(* TLS/PSK configuration *)
{attribute 'no_explicit_call':='Direct call not allowed for type FB_TlsConfig'}
{attribute 'no_assign'}
FUNCTION_BLOCK FB_TlsConfig
VAR
	_pskKey       : ARRAY[0..TCPADS_TLS_MAX_PSK_KEY_SIZE] OF BYTE;
	_pskKeyLen    : UDINT:=0;
	_sIdentity    : STRING(TCPADS_TLS_PSK_IDENTITY_SIZE);
	_sCaPath      : STRING(TCPADS_TLS_CERTIFICATE_PATH_SIZE);
	_sCrlPath     : STRING(TCPADS_TLS_CERTIFICATE_PATH_SIZE);
	_sCertPath    : STRING(TCPADS_TLS_CERTIFICATE_PATH_SIZE);
	_sKeyPath     : STRING(TCPADS_TLS_CERTIFICATE_PATH_SIZE);
	_sKeyPwd      : STRING(TCPADS_TLS_KEY_PASSWORD_SIZE);
	_listenFlags  : ST_TlsListenFlags:=DEFAULT_TLSLISTENFLAGS;
	_connectFlags : ST_TlsConnectFlags:=DEFAULT_TLSCONNECTFLAGS;
END_VAR

(* Adds CA certificate path *)
METHOD FINAL AddCa
VAR_INPUT
	sCaPath : STRING(TCPADS_TLS_CERTIFICATE_PATH_SIZE);
END_VAR
_sCaPath:=sCaPath;
END_METHOD

(* Adds certificate path *)
METHOD FINAL AddCert
VAR_INPUT
	sCertPath: STRING(TCPADS_TLS_CERTIFICATE_PATH_SIZE);
	sKeyPath: STRING(TCPADS_TLS_CERTIFICATE_PATH_SIZE);
	sKeyPwd: STRING(TCPADS_TLS_KEY_PASSWORD_SIZE);
END_VAR
_sCertPath:=sCertPath;
_sKeyPath:=sKeyPath;
_sKeyPwd:=sKeyPwd;
END_METHOD

METHOD FINAL AddConnectFlags
VAR_INPUT
	flags : ST_TlsConnectFlags;
END_VAR
_connectFlags:=flags;
END_METHOD

(* Adds certificate revocation list path *)
METHOD FINAL AddCrl
VAR_INPUT
	sCrlPath : STRING(TCPADS_TLS_CERTIFICATE_PATH_SIZE);
END_VAR
_sCrlPath:=sCrlPath;
END_METHOD

METHOD FINAL AddListenFlags
VAR_INPUT
	flags : ST_TlsListenFlags;
END_VAR
_listenFlags:=flags;
END_METHOD

(* Adds PSK and PSK identity *)
METHOD FINAL AddPsk
VAR_IN_OUT
	key : ARRAY[*] OF BYTE;
END_VAR
VAR_INPUT
	sIdentity : STRING(TCPADS_TLS_PSK_IDENTITY_SIZE);
END_VAR
_pskKeyLen:=MIN(DINT_TO_UDINT(UPPER_BOUND(key, 1) - LOWER_BOUND(key, 1) + 1), TCPADS_TLS_MAX_PSK_KEY_SIZE, SIZEOF(_pskKey));
MEMCPY(ADR(_pskKey[0]), ADR(key[LOWER_BOUND(key, 1)]), _pskKeyLen);
_sIdentity:=sIdentity;
END_METHOD

METHOD FINAL Clear
_sIdentity:='';
_pskKeyLen:=0;
MEMSET(ADR(_pskKey[0]), 0, SIZEOF(_pskKey));
_sCaPath:='';
_sCertPath:='';
_sKeyPath:='';
_sKeyPwd:='';
_sCrlPath:='';
END_METHOD

PROPERTY FINAL connectFlags : ST_TlsConnectFlags
GET
connectFlags:=_connectFlags;
END_GET
END_PROPERTY

PROPERTY FINAL listenFlags : ST_TlsListenFlags
GET
listenFlags:=_listenFlags;
END_GET
END_PROPERTY

(* Pointer to first PSK key byte *)
PROPERTY FINAL pskKey : PVOID
GET
pskKey:=SEL(_pskKeyLen = 0, ADR(_pskKey[0]), 0);
END_GET
END_PROPERTY

(* Byte size of PSK key *)
PROPERTY FINAL pskKeyLen : UDINT(0..TCPADS_TLS_MAX_PSK_KEY_SIZE)
GET
pskKeyLen:=_pskKeyLen;
END_GET
END_PROPERTY

(* CA certificate path *)
PROPERTY FINAL sCaPath : STRING(TCPADS_TLS_CERTIFICATE_PATH_SIZE)
GET
sCaPath:=_sCaPath;
END_GET
END_PROPERTY

(* Certificate path *)
PROPERTY FINAL sCertPath : STRING(TCPADS_TLS_CERTIFICATE_PATH_SIZE)
GET
sCertPath:=_sCertPath;
END_GET
END_PROPERTY

(* Certificate revocation list path *)
PROPERTY FINAL sCrlPath : STRING(TCPADS_TLS_CERTIFICATE_PATH_SIZE)
GET
sCrlPath:=_sCrlPath;
END_GET
END_PROPERTY

(* PSK key identity *)
PROPERTY FINAL sIdentity : STRING(TCPADS_TLS_PSK_IDENTITY_SIZE)
GET
sIdentity:=_sIdentity;
END_GET
END_PROPERTY

(* Certificate key path *)
PROPERTY FINAL sKeyPath : STRING(TCPADS_TLS_CERTIFICATE_PATH_SIZE)
GET
sKeyPath:=_sKeyPath;
END_GET
END_PROPERTY

(* Certificate key password *)
PROPERTY FINAL sKeyPwd : STRING(TCPADS_TLS_KEY_PASSWORD_SIZE)
GET
sKeyPwd:=_sKeyPwd;
END_GET
END_PROPERTY

END_FUNCTION_BLOCK

(* stored: Version 1.1.0.1
   POU FB_TlsConfig: Id {431216f2-1317-4e23-b121-71f1c6f4f3b0}, SpecialFunc None
   Method AddCa: Id {3f918c5b-c675-4c5d-8067-b5e641ad4391}
   Method AddCert: Id {b4df64f1-a1c6-4f62-bdce-0dd5195713bc}
   Method AddConnectFlags: Id {926e4460-d1ff-4890-afe0-63153b70e046}
   Method AddCrl: Id {e62f3fc2-fb79-4172-b635-04c32fa29160}
   Method AddListenFlags: Id {872e0c38-6839-4efd-affd-f4e34eab9833}
   Method AddPsk: Id {4892be68-e300-4c8a-bee6-417a151bc305}
   Method Clear: Id {5cf3987c-2f2d-4aa2-9d42-fc567e70b9cc}
   Property connectFlags: Id {d5ac45f6-4175-46d2-80a7-5d97502fcb40}
   Get Get: Id {a6df7a83-1dac-4c0c-8d86-d2e6d73344d6}
   Property listenFlags: Id {56b43e47-5dbf-4d79-90cc-0adddcfc7947}
   Get Get: Id {8e3a63f5-4283-4ad0-9198-ad2604cbb062}
   Property pskKey: Id {e6650675-d873-4375-b85f-11306b2e8e06}
   Get Get: Id {db17e43e-4d97-4824-b9ae-58053bcd1bad}
   Property pskKeyLen: Id {cd6a29bd-7b59-4d87-8190-08e7c531929f}
   Get Get: Id {2fbc4f9f-865b-4975-8f50-1ec98165e8ec}
   Property sCaPath: Id {ee747933-ca5f-4c91-b751-3139e7682da2}
   Get Get: Id {90112b83-b104-4d1c-975d-b3b421772ebf}
   Property sCertPath: Id {1fa9697f-ccb2-4934-aea8-2395138d4a6b}
   Get Get: Id {25b1eff8-efa0-4733-a8ba-e6cf8e182a95}
   Property sCrlPath: Id {921f265d-918b-4e9f-b2ed-d413b9c77288}
   Get Get: Id {e7344948-edda-4209-9f24-4e8c507f1ece}
   Property sIdentity: Id {c45a60b1-6670-46fb-9c14-e5b58619aec7}
   Get Get: Id {ec7517de-4959-4736-b3aa-788c203195f6}
   Property sKeyPath: Id {2855b108-7159-47ce-9f9c-be8ed43ba95f}
   Get Get: Id {04773564-daa5-40e8-80e9-7a329e5f4a65}
   Property sKeyPwd: Id {b5253c45-4680-427d-bd3c-936ded561d9f}
   Get Get: Id {58a73129-b41c-4dcc-95d7-0b8f7403ad2b} *)
